(* IEC 61131-3 sources: CodesysTest/export/Function Blocks/SolenoidValves/FB_SolenoidValve.pou, 1 file *)

(* ---- FB_SolenoidValve.pou.st ---- *)
(*#-#-#-#-#-#-#-#-#-#---Declaration---#-#-#-#-#-#-#-#-#-#-#-#-#*)

FUNCTION_BLOCK FB_SolenoidValve EXTENDS FB_BaseObject IMPLEMENTS ISolenoidValve, ISimulateable
VAR_INPUT
END_VAR
VAR_OUTPUT
	solenoid0 : BOOL;
	solenoid1 : BOOL;
END_VAR
VAR
	_simulateActive : BOOL;
END_VAR
(*#-#-#-#-#-#-#-#-#-#---Implementation---#-#-#-#-#-#-#-#-#-#-#-#-#*)
